{region '#Template'}
	{attribute 'Version' := '5.0.0.0'}
	{attribute 'Tags' := '"LCID": "1031", "Text": "RA, Beleuchtung, Aktor"'}
	{attribute 'Tags' := '"LCID": "1033", "Text": "RA, Lighting, Actuator"'}
	{attribute 'Using' := '"Type": "Template", "URI": "ST_BA_LightActuatorFeedback"'}
	{attribute 'Description' := '"LCID": "1031", "Text": "Beleuchtung Analogaktor"'}
	{attribute 'Description' := '"LCID": "1033", "Text": "Lighting analog-actuator"'}
{endregion}
FUNCTION_BLOCK FB_BA_LightAnalog  EXTENDS FB_BA_View

VAR_INPUT
	bEn						: BOOL;						// FB-enable 
	stLightingCmd			: ST_BA_Lighting;   		// command-structure
END_VAR
VAR_OUTPUT
	fActualLightValue		: REAL;						// actual light value
	eActualLightPrio		: BYTE;						// actual telegram priority
	stFeedback				: ST_BA_LightActuatorFeedback;
END_VAR
VAR_INPUT CONSTANT				 
	ActualLightValue		: FB_BA_AO_Raw;
END_VAR
VAR
	nLgtVal 		AT %Q*	: INT;
END_VAR
VAR // added by the converter: edge detectors and wires of the graphical bodies
    _s1 : ST_BA_LightActuatorFeedback;
END_VAR

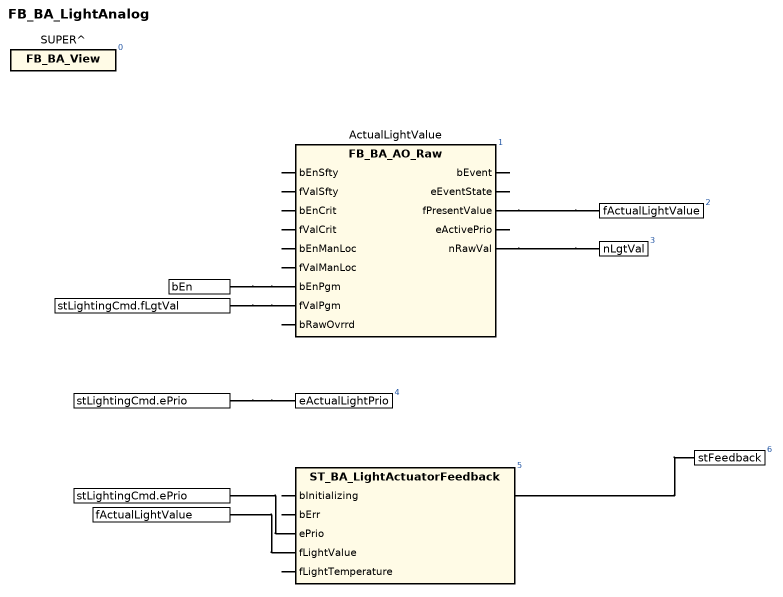
SUPER^(); // FB_BA_View
ActualLightValue(bEnPgm := bEn, fValPgm := stLightingCmd.fLgtVal); // FB_BA_AO_Raw
fActualLightValue := ActualLightValue.fPresentValue;
nLgtVal := ActualLightValue.nRawVal;
eActualLightPrio := stLightingCmd.ePrio;
// compose _s1 : ST_BA_LightActuatorFeedback
_s1.ePrio := stLightingCmd.ePrio;
_s1.fLightValue := fActualLightValue;
stFeedback := _s1;

METHOD FB_init : BOOL
VAR_INPUT
	bInitRetains : BOOL; // if TRUE; the retain variables are initialized (warm start / cold start)
	bInCopyCode : BOOL;  // if TRUE; the instance afterwards gets moved into the copy code (online change)
END_VAR

{region 'BACnet'}
ActualLightValue.iParent					:= THIS^;
ActualLightValue.iLabel						:= LblFun_FeedbackLightValue;  
ActualLightValue.eUnit						:= E_BA_Unit.eOther_Percent;
ActualLightValue.fResolution 				:= 0.003051851;					// 100% -> 32767
ActualLightValue.fScaleOffset 				:= 0;
ActualLightValue.fCOVIncrement				:= BA2_Param.fDefCOVIncrement;
ActualLightValue.bEnManualRm				:= FALSE;	//	Priority  8	
ActualLightValue.fValManualRm				:= 0.0;		//	Priority  8
ActualLightValue.nEventClassID				:= EC_ID.NC80;
ActualLightValue.stTimeDelay.nToNormal		:= BA2_Param.nDefTimeDelay_ToNormal;
ActualLightValue.stTimeDelay.nToAbnormal	:= BA2_Param.nDefTimeDelay_ToAbnormal;
ActualLightValue.stHighLimit.bEnable		:= FALSE;
ActualLightValue.stHighLimit.fValue			:= 0.0;		
ActualLightValue.stLowLimit.bEnable			:= FALSE;
ActualLightValue.stLowLimit.fValue			:= 0.0;
ActualLightValue.fLimitDeadband 			:= BA2_Param.fDefLimitDeadband;
ActualLightValue.aEventTransitionText[1]	:= txtEvent_Disturb;
ActualLightValue.aEventTransitionText[2]	:= txtEvent_None;
ActualLightValue.aEventTransitionText[3]	:= txtEvent_Normal;
ActualLightValue.bEventDetectionEnable		:= FALSE;
ActualLightValue.eEnPlantLock				:= E_BA_LockPriority.eNoLock;		
{endregion}
END_METHOD

END_FUNCTION_BLOCK

(* stored: Version 1.1.0.1, ProductVersion 3.1.4024.12
   POU FB_BA_LightAnalog: Id {9de46ba0-22b3-45ea-ad9f-500acf2cfb1f}, SpecialFunc None
   Method FB_init: Id {15b22bcd-9302-4971-8a20-55c796f68aad} *)
